// TwinCAT 3 PLC project cpu
// ProgramVersion: 3.1.4024.0
// libraries:
//   Tc2_Standard, * (Beckhoff Automation GmbH)
//   Tc2_System, * (Beckhoff Automation GmbH)
//   Tc3_Module, * (Beckhoff Automation GmbH)
// project tree:
//   DUTs/ ISensor.TcIO
//   GVLs/ IO.TcGVL
//   / MAIN.TcPOU, PlcTask.TcTTO
//   POUs/Sensor/DUT/ SensorBeckhoffIO_In.TcDUT
//   POUs/Sensor/ SensorBeckhoff.TcPOU
//   POUs/ transform.TcPOU, VFD.TcPOU
// real-time tasks:
//   TASK PlcTask: cycle T#10ms, priority 20, ADS port 350

CONFIGURATION cpu
    RESOURCE PLC ON TwinCAT3
        TASK PlcTask(INTERVAL := T#10ms, PRIORITY := 20);
        PROGRAM MAIN WITH PlcTask : MAIN;
    END_RESOURCE
END_CONFIGURATION

// ---- POUs/Sensor/DUT/SensorBeckhoffIO_In.TcDUT
TYPE SensorBeckhoffIO_In :
	STRUCT
		ValuesRaw 		: INT;
	END_STRUCT
END_TYPE

// ---- GVLs/IO.TcGVL
{attribute 'qualified_only'}
VAR_GLOBAL
	sensorPoti		AT %I*	: SensorbeckhoffIO_In;
END_VAR

// ---- DUTs/ISensor.TcIO
INTERFACE ISensor

PROPERTY Value : LREAL
GET
END_GET
END_PROPERTY

END_INTERFACE

// ---- MAIN.TcPOU
PROGRAM MAIN
VAR
	poti 	: SensorBeckhoff(IO.sensorPoti, 0, 32767, 0, 1);
	vfd		: VFD;
	
	choice	: DINT := 1;
END_VAR

poti.update();
vfd.update();	

		
CASE choice OF
	1: 	// run motor with 10% of SpeedMax and variable torque
		vfd.executeOperation(0.1, poti.Value);
		
	2:	// run motor with varibale speed and 100% torque
		vfd.executeOperation(poti.Value, 1);
	
END_CASE

END_PROGRAM

// ---- POUs/Sensor/SensorBeckhoff.TcPOU
{attribute 'no_explicit_call' := 'do not call this POU directly'} 
FUNCTION_BLOCK SensorBeckhoff IMPLEMENTS ISensor, __SYSTEM.IQueryInterface
VAR
	io_in			: REFERENCE TO SensorBeckhoffIO_in;
	_value			: LREAL;
	
	inputMin		: LREAL;
	inputMax		: LREAL;
	outputMin		: LREAL;
	outputMax		: LREAL;
END_VAR

METHOD FB_init : BOOL
VAR_INPUT
	bInitRetains : BOOL; // if TRUE, the retain variables are initialized (warm start / cold start)
	bInCopyCode : BOOL;  // if TRUE, the instance afterwards gets moved into the copy code (online change)
	IO_in			: REFERENCE TO SensorBeckhoffIO_in;
	InputMin		: LREAL;
	InputMax		: LREAL;
	OutputMin		: LREAL;
	OutputMax		: LREAL;
END_VAR
THIS^.io_in REF= IO_in;
THIS^.inputMin := InputMin;
THIS^.inputMax := InputMax;
THIS^.outputMin := OutputMin;
THIS^.outputMax := OutputMax;
END_METHOD

METHOD update : BOOL
_value := transform(TO_LREAL(io_in.ValuesRaw), inputMin, inputMax, outputMin, outputMax, LimitY := TRUE);
END_METHOD

PROPERTY Value : LREAL
GET
Value := _value;
END_GET
END_PROPERTY

END_FUNCTION_BLOCK

// ---- POUs/transform.TcPOU
(*
	This function transform X range to a Y range, with the option of limiting 
	the output Y.
*)
FUNCTION transform : LREAL
VAR_INPUT
	Value		: LREAL;
	X1			: LREAL;
	X2			: LREAL;
	Y1			: LREAL;
	Y2			: LREAL;
	LimitY		: BOOL;
END_VAR
VAR
END_VAR

IF X2 - X1 <> 0 THEN
	transform := (Y2 - Y1) / (X2 - X1) * (Value - X1) + Y1;
	IF LimitY THEN
		IF Y2 >= Y1 THEN 
			transform := LIMIT(Y1, transform, Y2);
		ELSE
			transform := LIMIT(Y2, transform, Y1);			
		END_IF
	END_IF
ELSE
	transform := 0;
END_IF

END_FUNCTION

// ---- POUs/VFD.TcPOU
{attribute 'no_explicit_call' := 'do not call this POU directly'} 
FUNCTION_BLOCK VFD
VAR
END_VAR

METHOD executeOperation : BOOL
VAR_INPUT
	SpeedRel 	: LREAL;
	TorqueRel	: LREAL;
END_VAR
END_METHOD

PROPERTY Speed : LREAL
GET
END_GET
END_PROPERTY

PROPERTY SpeedMax : LREAL
GET
END_GET
END_PROPERTY

PROPERTY Torque : LREAL
GET
END_GET
END_PROPERTY

PROPERTY TorqueMax : LREAL
GET
END_GET
END_PROPERTY

PROPERTY TorqueRel : LREAL
GET
END_GET
END_PROPERTY

METHOD update : BOOL
VAR_INPUT
END_VAR
END_METHOD

END_FUNCTION_BLOCK
